PROGRAM MAIN
VAR
END_VAR

END_PROGRAM

(* stored: Version 1.1.0.1, ProductVersion 3.1.0.38
   POU MAIN: Id {87daacfd-dd5b-456b-afd6-541cb130f9ba}, SpecialFunc None *)
